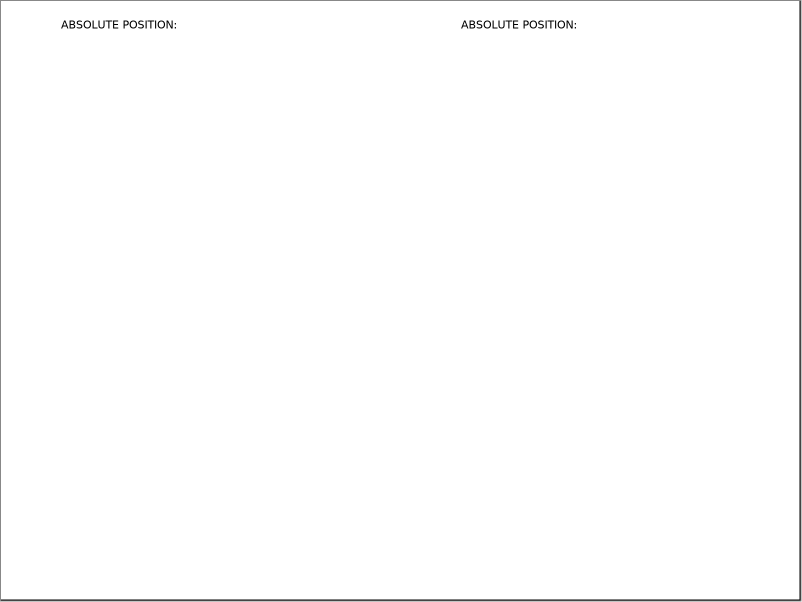
VISUALIZATION F44_Halt_Phasing  // 802x602
    Rectangle (0,0 800x600)
    Label (10,10 170x30), "ABSOLUTE POSITION:"
    Label (410,10 170x30), "ABSOLUTE POSITION:"
END_VISUALIZATION

(* stored: Version 1.1.0.1, ProductVersion 3.1.4022.7
   Visu F44_Halt_Phasing: Id {1daf95aa-8623-464d-b416-afa8f3ad3ffe} *)
